SYSTEM Test_12 (* System Configuration *)
  (* Standard: 61499-1 *)
  (* Version 0.3, 2003-12-05, JHC, Rockwell Automation, Renamed from NEWSYSTEM. *)
  (* Version 0.2, 2002-11-05, JHC, Rockwell Automation, Fixed missing (empty) FBD in Application. *)
  (* Version 0.1, 2002-01-17, JHC, Rockwell Automation, Minor cleanup *)
  (* Version 0.0, 2000-05-27, JHC, Rockwell Automation *)
  APPLICATION APP1
  END_APPLICATION
  DEVICE WORKERS_HMI : FRAME_DEVICE(BOUNDS := [300,300,800,500], GRID := [1,1])
    RESOURCE Worker1 : PANEL_RESOURCE(ROWS := 4, COLS := 2)
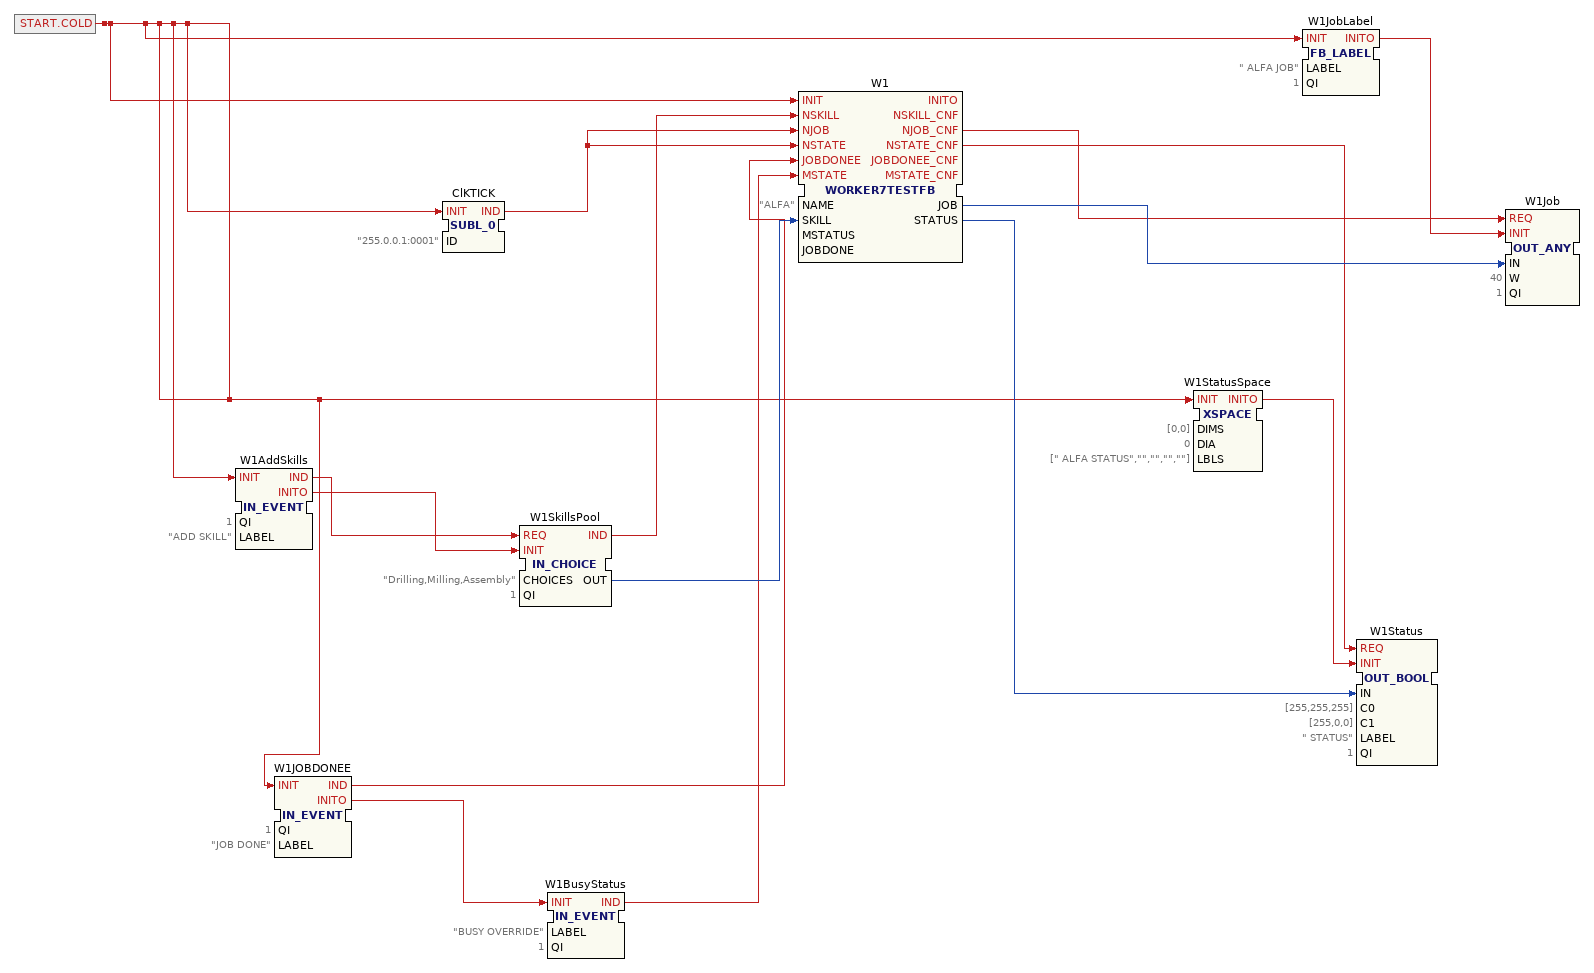
      FBS
        W1 : WORKER7TESTFB(NAME := "ALFA");
        W1SkillsPool : IN_CHOICE(CHOICES := "Drilling,Milling,Assembly", QI := 1);
        W1AddSkills : IN_EVENT(QI := 1, LABEL := "ADD SKILL");
        W1Status : OUT_BOOL(C0 := [255,255,255], C1 := [255,0,0], LABEL := "        STATUS", QI := 1);
        W1Job : OUT_ANY(W := 40, QI := 1);
        W1JobLabel : FB_LABEL(LABEL := "        ALFA JOB", QI := 1);
        W1StatusSpace : XSPACE(DIMS := [0,0], DIA := 0, LBLS := ["        ALFA STATUS","","","",""]);
        ClKTICK : SUBL_0(ID := "255.0.0.1:0001");
        W1JOBDONEE : IN_EVENT(QI := 1, LABEL := "JOB DONE");
        W1BusyStatus : IN_EVENT(LABEL := "BUSY OVERRIDE", QI := 1);
      END_FBS
      EVENT_CONNECTIONS
        START.COLD TO W1.INIT;
        W1SkillsPool.IND TO W1.NSKILL;
        W1AddSkills.IND TO W1SkillsPool.REQ;
        W1.NSTATE_CNF TO W1Status.REQ;
        W1.NJOB_CNF TO W1Job.REQ;
        START.COLD TO W1JobLabel.INIT;
        W1JobLabel.INITO TO W1Job.INIT;
        START.COLD TO W1StatusSpace.INIT;
        W1StatusSpace.INITO TO W1Status.INIT;
        START.COLD TO W1AddSkills.INIT;
        W1AddSkills.INITO TO W1SkillsPool.INIT;
        START.COLD TO ClKTICK.INIT;
        ClKTICK.IND TO W1.NJOB;
        ClKTICK.IND TO W1.NSTATE;
        W1JOBDONEE.IND TO W1.JOBDONEE;
        START.COLD TO W1JOBDONEE.INIT;
        W1JOBDONEE.INITO TO W1BusyStatus.INIT;
        W1BusyStatus.IND TO W1.MSTATE;
      END_CONNECTIONS
      DATA_CONNECTIONS
        W1SkillsPool.OUT TO W1.SKILL;
        W1.JOB TO W1Job.IN;
        W1.STATUS TO W1Status.IN;
      END_CONNECTIONS
    END_RESOURCE
    RESOURCE Worker2 : PANEL_RESOURCE(ROWS := 4, COLS := 2)
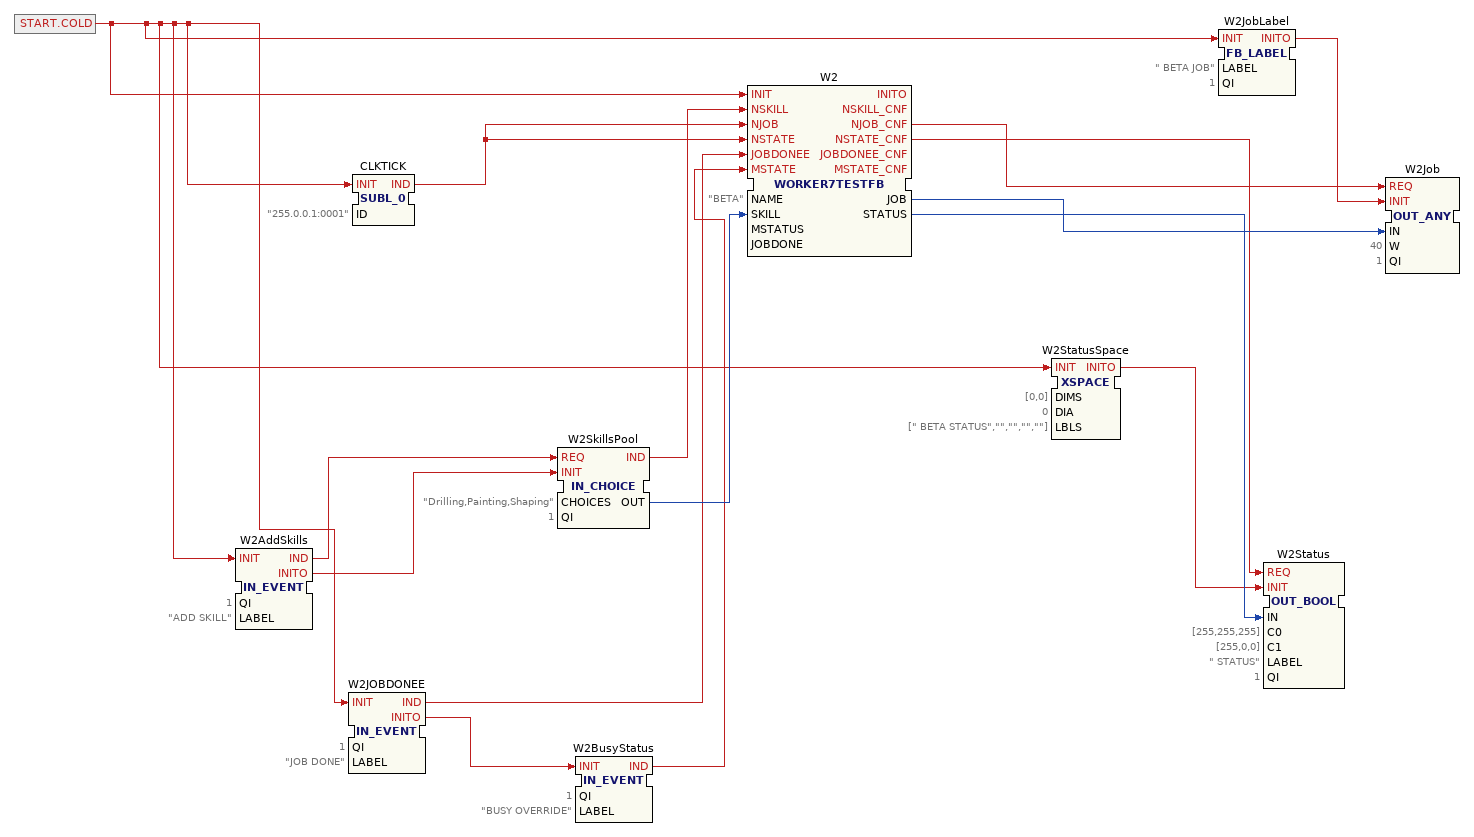
      FBS
        W2 : WORKER7TESTFB(NAME := "BETA");
        W2SkillsPool : IN_CHOICE(CHOICES := "Drilling,Painting,Shaping", QI := 1);
        W2AddSkills : IN_EVENT(QI := 1, LABEL := "ADD SKILL");
        W2Status : OUT_BOOL(C0 := [255,255,255], C1 := [255,0,0], LABEL := "        STATUS", QI := 1);
        W2Job : OUT_ANY(W := 40, QI := 1);
        W2JobLabel : FB_LABEL(LABEL := "        BETA JOB", QI := 1);
        W2StatusSpace : XSPACE(DIMS := [0,0], DIA := 0, LBLS := ["        BETA STATUS","","","",""]);
        CLKTICK : SUBL_0(ID := "255.0.0.1:0001");
        W2JOBDONEE : IN_EVENT(QI := 1, LABEL := "JOB DONE");
        W2BusyStatus : IN_EVENT(QI := 1, LABEL := "BUSY OVERRIDE");
      END_FBS
      EVENT_CONNECTIONS
        START.COLD TO W2.INIT;
        W2SkillsPool.IND TO W2.NSKILL;
        W2AddSkills.IND TO W2SkillsPool.REQ;
        W2.NSTATE_CNF TO W2Status.REQ;
        W2.NJOB_CNF TO W2Job.REQ;
        START.COLD TO W2JobLabel.INIT;
        W2JobLabel.INITO TO W2Job.INIT;
        START.COLD TO W2StatusSpace.INIT;
        W2StatusSpace.INITO TO W2Status.INIT;
        START.COLD TO W2AddSkills.INIT;
        W2AddSkills.INITO TO W2SkillsPool.INIT;
        START.COLD TO CLKTICK.INIT;
        CLKTICK.IND TO W2.NJOB;
        CLKTICK.IND TO W2.NSTATE;
        START.COLD TO W2JOBDONEE.INIT;
        W2JOBDONEE.IND TO W2.JOBDONEE;
        W2JOBDONEE.INITO TO W2BusyStatus.INIT;
        W2BusyStatus.IND TO W2.MSTATE;
      END_CONNECTIONS
      DATA_CONNECTIONS
        W2SkillsPool.OUT TO W2.SKILL;
        W2.JOB TO W2Job.IN;
        W2.STATUS TO W2Status.IN;
      END_CONNECTIONS
    END_RESOURCE
  END_DEVICE
  DEVICE GLOBAL_CONTROLLER : FRAME_DEVICE(BOUNDS := [800,800,150,150], GRID := [1,1])
    RESOURCE GlobalClock : PANEL_RESOURCE(ROWS := 0, COLS := 0)
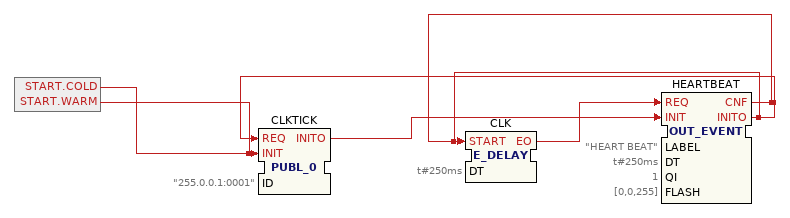
      FBS
        CLKTICK : PUBL_0(ID := "255.0.0.1:0001");
        HEARTBEAT : OUT_EVENT(LABEL := "HEART BEAT", DT := t#250ms, QI := 1, FLASH := [0,0,255]);
        CLK : E_DELAY(DT := t#250ms);
      END_FBS
      EVENT_CONNECTIONS
        CLK.EO TO HEARTBEAT.REQ;
        HEARTBEAT.CNF TO CLK.START;
        HEARTBEAT.CNF TO CLKTICK.REQ;
        START.COLD TO CLKTICK.INIT;
        START.WARM TO CLKTICK.INIT;
        CLKTICK.INITO TO HEARTBEAT.INIT;
        HEARTBEAT.INITO TO CLK.START;
        HEARTBEAT.INITO TO CLKTICK.REQ;
      END_CONNECTIONS
    END_RESOURCE
  END_DEVICE
  DEVICE ROBOT_CONTROLLER : FRAME_DEVICE(GRID := [1,1], BOUNDS := [1100,300,600,400])
    RESOURCE ROBOT : PANEL_RESOURCE(ROWS := 7, COLS := 2)
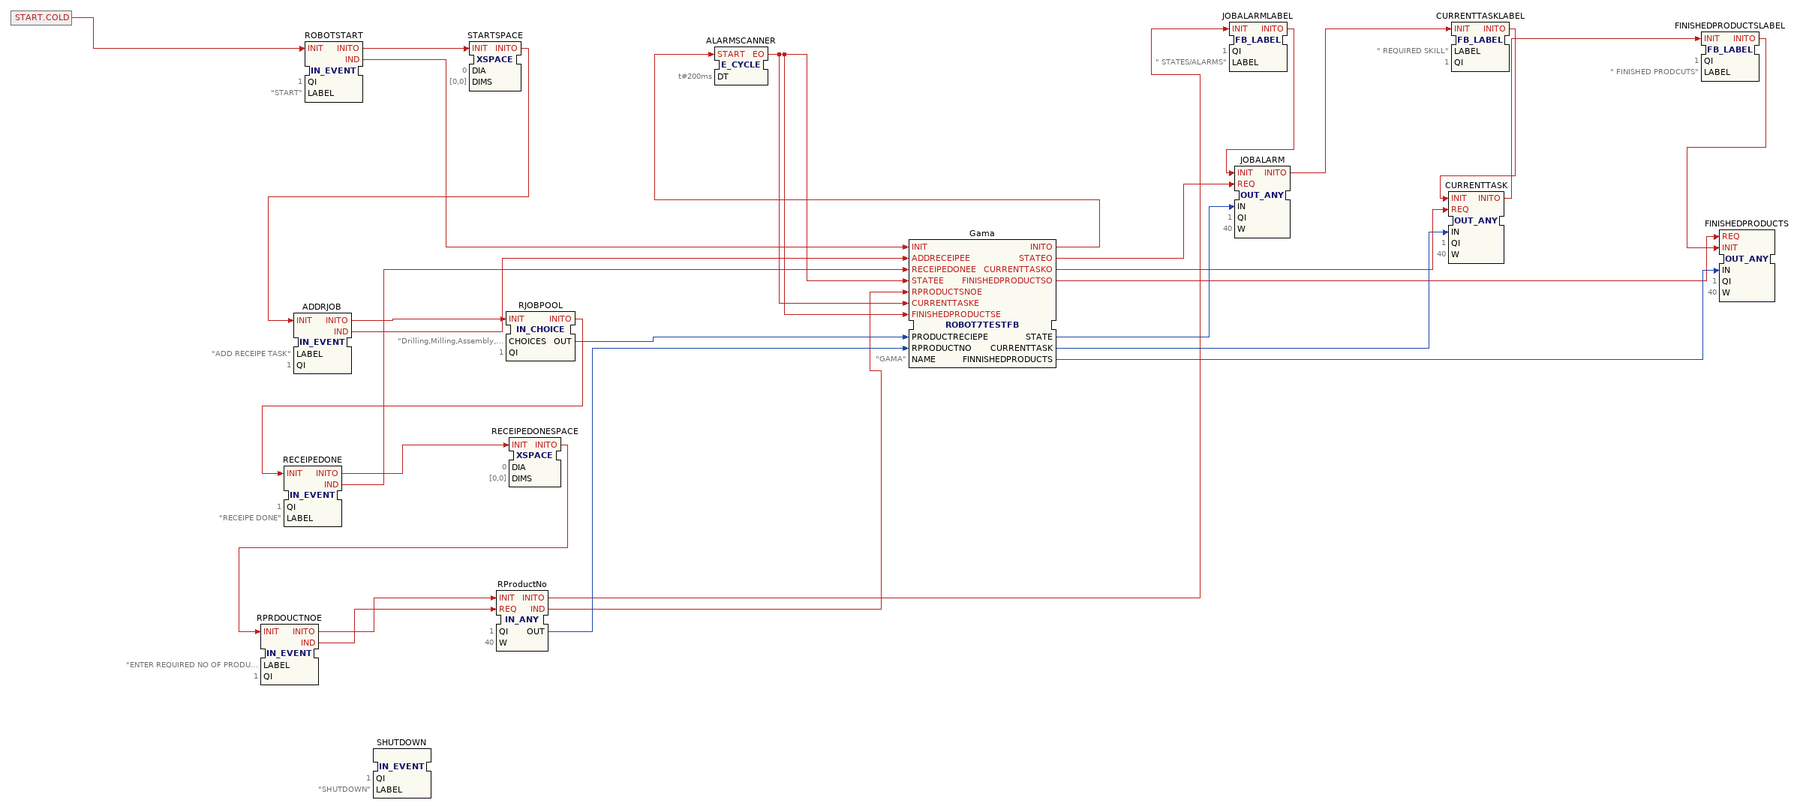
      FBS
        Gama : ROBOT7TESTFB(NAME := "GAMA");
        ROBOTSTART : IN_EVENT(QI := 1, LABEL := "START");
        ADDRJOB : IN_EVENT(LABEL := "ADD RECEIPE TASK", QI := 1);
        RJOBPOOL : IN_CHOICE(CHOICES := "Drilling,Milling,Assembly,Painting,Shaping", QI := 1);
        JOBALARM : OUT_ANY(QI := 1, W := 40);
        JOBALARMLABEL : FB_LABEL(QI := 1, LABEL := "                                  STATES/ALARMS");
        ALARMSCANNER : E_CYCLE(DT := t#200ms);
        STARTSPACE : XSPACE(DIA := 0, DIMS := [0,0]);
        SHUTDOWN : IN_EVENT(QI := 1, LABEL := "SHUTDOWN");
        RECEIPEDONE : IN_EVENT(QI := 1, LABEL := "RECEIPE DONE");
        RECEIPEDONESPACE : XSPACE(DIA := 0, DIMS := [0,0]);
        RPRDOUCTNOE : IN_EVENT(LABEL := "ENTER REQUIRED NO OF PRODUCTS", QI := 1);
        RProductNo : IN_ANY(QI := 1, W := 40);
        CURRENTTASKLABEL : FB_LABEL(LABEL := "                                   REQUIRED SKILL", QI := 1);
        CURRENTTASK : OUT_ANY(QI := 1, W := 40);
        FINISHEDPRODUCTSLABEL : FB_LABEL(QI := 1, LABEL := "                               FINISHED PRODCUTS");
        FINISHEDPRODUCTS : OUT_ANY(QI := 1, W := 40);
      END_FBS
      EVENT_CONNECTIONS
        ADDRJOB.INITO TO RJOBPOOL.INIT;
        JOBALARMLABEL.INITO TO JOBALARM.INIT;
        START.COLD TO ROBOTSTART.INIT;
        STARTSPACE.INITO TO ADDRJOB.INIT;
        ROBOTSTART.INITO TO STARTSPACE.INIT;
        ROBOTSTART.IND TO Gama.INIT;
        Gama.INITO TO ALARMSCANNER.START;
        ADDRJOB.IND TO Gama.ADDRECEIPEE;
        RJOBPOOL.INITO TO RECEIPEDONE.INIT;
        RECEIPEDONE.INITO TO RECEIPEDONESPACE.INIT;
        RECEIPEDONE.IND TO Gama.RECEIPEDONEE;
        ALARMSCANNER.EO TO Gama.STATEE;
        RPRDOUCTNOE.INITO TO RProductNo.INIT;
        RProductNo.INITO TO JOBALARMLABEL.INIT;
        RECEIPEDONESPACE.INITO TO RPRDOUCTNOE.INIT;
        RPRDOUCTNOE.IND TO RProductNo.REQ;
        RProductNo.IND TO Gama.RPRODUCTSNOE;
        JOBALARM.INITO TO CURRENTTASKLABEL.INIT;
        CURRENTTASKLABEL.INITO TO CURRENTTASK.INIT;
        Gama.STATEO TO JOBALARM.REQ;
        Gama.CURRENTTASKO TO CURRENTTASK.REQ;
        CURRENTTASK.INITO TO FINISHEDPRODUCTSLABEL.INIT;
        Gama.FINISHEDPRODUCTSO TO FINISHEDPRODUCTS.REQ;
        FINISHEDPRODUCTSLABEL.INITO TO FINISHEDPRODUCTS.INIT;
        ALARMSCANNER.EO TO Gama.CURRENTTASKE;
        ALARMSCANNER.EO TO Gama.FINISHEDPRODUCTSE;
      END_CONNECTIONS
      DATA_CONNECTIONS
        RJOBPOOL.OUT TO Gama.PRODUCTRECIEPE;
        Gama.STATE TO JOBALARM.IN;
        RProductNo.OUT TO Gama.RPRODUCTNO;
        Gama.CURRENTTASK TO CURRENTTASK.IN;
        Gama.FINNISHEDPRODUCTS TO FINISHEDPRODUCTS.IN;
      END_CONNECTIONS
    END_RESOURCE
  END_DEVICE
END_SYSTEM
